Universal Robots PolyScope program: APS2Socket.urp

Program APS2Socket (installation=default directory=/programs/APS2OsUltimosRomanticos createdIn=3.15.3.106223 lastSavedIn=3.15.3.106223 robotSerialNumber=2017357017)
Calibrated DH parameters: a=[0.0001, -0.032836, -0.39033, 0.000086, 0.000053, 0]; d=[0.089393, 264.548863, -261.578988, -2.85966, 0.094927, 0.082356]; alpha=[1.569373, -0.001603, 0.013671, 1.570599, -1.570158, 0]; deltaTheta=[0.000031, -1.49356, 1.597104, -0.103695, -0.000023, -0.000043]
BeforeStart
  SocketIP := socket_open("10.103.16.140",30000)
  MoveJ speed 60 deg/s, acceleration 80 deg/s^2 (useActiveTCP=true)
    Waypoint Waypoint_1: TCP in base x=63.867 y=-618.041 z=296.078 mm, rx=0.0391 ry=-0.003 rz=0.1194 rad; joints [85.759, -70.576, 59.854, -77.008, -89.434, -11.122] deg; flange x=64.028 y=-625.06 z=475.941 mm, rx=-0.1873 ry=3.134 rz=0.0612 rad
Robot Program (runOnlyOnce=false)
  Loop While (checkContinuously=false) expression=SocketIP≟ False
    SocketIP := socket_open("10.103.16.140",30000)
    Wait Sleep waitTime=0.5
  Script: socket_send_string("asking_for_data")
  Wait Sleep waitTime=0.5
  read_ascii := socket_read_ascii_float(3)
  Wait Sleep waitTime=0.5
  SocketIP := False
  Script: socket_close()
  If read_ascii[0]≠0
    pose_desejada := p[read_ascii[1]/1000,read_ascii[2]/1000,0,0,0,d2r(90)]
    pose_atual := get_actual_tcp_pose()
    trans_pose := pose_trans(pose_atual,pose_desejada)
    MoveL speed 250 mm/s, acceleration 1200 mm/s^2 (useActiveTCP=true) feature=Base
      Waypoint Waypoint (Variable): variable=trans_pose
      Wait Sleep waitTime=0.5
      Waypoint Waypoint_1: TCP in base x=63.867 y=-618.041 z=296.078 mm, rx=0.0391 ry=-0.003 rz=0.1194 rad; joints [85.759, -70.576, 59.854, -77.008, -89.434, -11.122] deg; flange x=64.028 y=-625.06 z=475.941 mm, rx=-0.1873 ry=3.134 rz=0.0612 rad
